{attribute 'qualified_only'}
// ------------------------------------------------------------------------- 
//  SRCI Robot Library                                                
// ------------------------------------------------------------------------- 
//                                                                           
//  Object:      RiState                                       
//  Author:      Thorsten Brach                                                
//  Date:        2024-06-01
//
//  Description:                                              
//   
//                                                                           
//  Copyright: 
//    (C) 2024 Thorsten Brach. All rights reserved                                                                                                                                            
//             Licensed under the MIT License.
//                                                                           
//  Disclaimer:                                                                           
//    This project is provided without any guarantee and can be used for   
//    private and commercial purposes. Any use is at the user’s 
//    own risk and responsibility.
//
// -------------------------------------------------------------------------
TYPE RiState :
(
  /// RI is not initialized
  NOT_INITIALIZED := 0,
  /// Initialization finished successfully
  INITIALIZED := 1,
  /// Data between RC and PLC has been synchronized
  SYNCHRONIZED := 2
)USINT;
END_TYPE

{attribute 'qualified_only'}
TYPE TelegramState :
(
  /// Default
  UNDEFINED := 0,
  /// Telegram control does not match the telegram state
  ERROR_161_TELEGRAM_CONTROL_MISMATCH_TELEGRAM_STATE := 161,
  /// Initialization lost for unknown reason. See message log after reinitializing
  ERROR_162_INIT_LOST_UNKNOWN := 162,
  /// Telegram length does not match the length provided in the communication interface.
  ERROR_163_TELEGRAM_LENGTH_MISMATCH := 163,
  /// Incompatible major SRCI version
  ERROR_164_SRCI_MAJOR_VERSION_INCOMPATIBLE := 164,
  /// Lifesign timeout
  ERROR_165_LIFESIGN_TIMEOUT := 165,
  /// The selected optional cyclic data does not fit in the given telegram size
  ERROR_166_CYCLIC_DATA_TOO_LARGE := 166,
  /// The robot interface was reset after being initialized
  ERROR_167_INTERFACE_WAS_RESET_AFTER_INIT := 167,
  /// Telegram sequence timeout
  ERROR_168_TELEGRAM_SEQ_TIMEOUT := 168,
  /// The telegram number changed after initialization
  ERROR_169_TELEGRAM_NO_CHANGED_AFTER_INIT := 169,
  /// Invalid AxesGroupID
  ERROR_170_AXESGROUP_ID_INVALID := 170,
  /// Telegram number is invalid. E.g. TwoSequences is only activated in one direction
  ERROR_171_TELEGRAM_NUMBER_INVALID := 171,
  /// Telegram Number is not supported
  ERROR_172_TELEGRAM_NUMBER_NOT_SUPPORTED := 172,
  /// Server connection lost
  ERROR_173_SERVER_CONNECTION_LOST := 173,
  /// The RC is currently not initialized but has state in the ACR
  READY_TO_RESUME := 253,
  /// The RC is currently not initialized and has no state in the ACR
  READY_FOR_INITIALIZATION := 254,
  /// The RC state is Initialized
  INITIALIZED := 255  
)USINT;
END_TYPE

{attribute 'qualified_only'}
// ------------------------------------------------------------------------- 
//  SRCI Robot Library                                                
// ------------------------------------------------------------------------- 
//                                                                           
//  Object:      AreaType                                       
//  Author:      Thorsten Brach                                                
//  Date:        2024-06-01
//
//  Description:                                              
//   
//                                                                           
//  Copyright: 
//    (C) 2024 Thorsten Brach. All rights reserved                                                                                                                                            
//             Licensed under the MIT License.
//                                                                           
//  Disclaimer:                                                                           
//    This project is provided without any guarantee and can be used for   
//    private and commercial purposes. Any use is at the user’s 
//    own risk and responsibility.
//
// -------------------------------------------------------------------------
TYPE AreaType :
(
  /// 0: Axes
  AXES := 0,
  /// 1: Box (default)
  BOX := 1,
  /// 2: Cylinder
  CYLINDER := 2,
  /// 3: Sphere (only DefinitionMode 1)
  SPHERE := 3
)USINT;
END_TYPE

{attribute 'qualified_only'}
// ------------------------------------------------------------------------- 
//  SRCI Robot Library                                                
// ------------------------------------------------------------------------- 
//                                                                           
//  Object:      AxesGroupParameterCmdEntries                                       
//  Author:      Thorsten Brach                                                
//  Date:        2024-06-01
//
//  Description:                                              
//   
//                                                                           
//  Copyright: 
//    (C) 2024 Thorsten Brach. All rights reserved                                                                                                                                            
//             Licensed under the MIT License.
//                                                                           
//  Disclaimer:                                                                           
//    This project is provided without any guarantee and can be used for   
//    private and commercial purposes. Any use is at the user’s 
//    own risk and responsibility.
//
// -------------------------------------------------------------------------
TYPE AxesGroupParameterCmdEntries :
(
  /// Handles multiple mechanisms required for operation of the interface
  RobotTask := 0, // No function code  
  /// Read robot-specific data from the RC
  ReadRobotData := 9002,  
  /// Enable/Disable robot into RA power state "Enabled"
  EnableRobot := 1,  
  /// Acknowledgement all pending errors
  GroupReset := 2,  
  /// Read the actual position – TCP: X…RZ + config/Turn, Joint: (J1…E6)
  ReadActualPosition := 3,
  /// Read the actual position cyclically
  ReadActualPositionCyclic := 4,   
  /// Read D-H-parameters of robot
  ReadDHParameter := 5,  
  /// Restart/reboot of the RC
  RestartController := 6,  
  /// Read actual TCP velocity
  ReadActualTCPVelocity := 7,  
  /// Login on RC from PLC
  UserLogin := 8,  
  /// Switch language of robot teach pendant from PLC
  SwitchLanguage := 9,  
  /// Reads and writes specific configuration parameters on RC that are required for the RI to work
  ExchangeConfiguration := 10,  
  /// Set active sequence
  SetSequence := 11,  
  /// Change actual speed override
  ChangeSpeedOverride := 12,  
  /// Read error codes of pending errors and move them into user data block "RobotData"
  ReadMessages := 13,  
  /// Read reference values of robot dynamics for path movement
  ReadRobotReferenceDynamics := 14,  
  /// Change configuration of selected user frame number
  WriteFrameData := 15,  
  /// Change configuration of selected tool number
  WriteToolData := 16,  
  /// Change configuration of selected payload number
  WriteLoadData := 17,  
  /// Write reference values of robot dynamics for path movement
  WriteRobotReferenceDynamics := 18,  
  /// Write default values of dynamic parameters used by move commands
  WriteRobotDefaultDynamics := 19,  
  /// Read default values of dynamic parameters used by move commands
  ReadRobotDefaultDynamics := 20,  
  /// Read content of selected user frame number
  ReadFrameData := 21,  
  /// Read content of selected tool number
  ReadToolData := 22,  
  /// Read content of selected payload number
  ReadLoadData := 23,  
  /// Read actual software limits of the axes Positive and negative Limit of Joint J1…J6, E1…E6
  ReadRobotSWLimits := 24,  
  /// Change robot limits of robot axes (degree)
  WriteRobotSWLimits := 25,  
  /// Switch operation mode of RC (Automatic External, T1 External, T2 External)
  SetOperationMode := 26,  
  /// Read configuration of defined work areas
  ReadWorkArea := 27,  
  /// Define work area
  WriteWorkArea := 28,  
  /// Enable/Disable work areas of RC and check if TCP is inside/outside of active work area
  ActivateWorkArea := 29,  
  /// Monitor enabled work areas
  MonitorWorkArea := 30,  
  /// Jog robot manually
  GroupJog := 31,  
  /// Move the TCP to an absolute cartesian position (linear interpolation)
  MoveLinearAbsolute := 32,  
  /// Move Joints to an absolute cartesian position (Absolute cartesian PTP) (Joint interpolated movement)
  MoveDirectAbsolute := 33,  
  /// Move all joints to an absolute joint position (Absolute Joint PTP)
  MoveAxesAbsolute := 34,  
  /// Abort actual movement and delete buffer
  GroupStop := 35,  
  /// Interrupt active movement, possible to continue movement
  GroupInterrupt := 36,  
  /// Continue interrupted path
  GroupContinue := 37,  
  /// Move the TCP relative to the actual cartesian position (linear interpolation)
  MoveLinearRelative := 38,  
  /// Move Joints relative to relative cartesian position (Relative cartesian PTP) (Joint interpolated movement)
  MoveDirectRelative := 39,  
  /// Move all joints relative to actual joint position (Relative Joint PTP)
  MoveAxesRelative := 40,  
  /// Return to path left during active interrupt
  ReturnToPrimary := 41,  
  /// Move the TCP to an absolute joint position (linear interpolation)
  MoveCircularAbsolute := 42,  
  /// Move the TCP relative to the actual cartesian position (circular interpolation)
  MoveCircularRelative := 43,  
  /// Move the TCP relative to a reference cartesian position (linear interpolation)
  MoveLinearOffset := 44,  
  /// Move the TCP relative to a reference cartesian position (PTPT interpolation)
  MoveDirectOffset := 45,  
  /// Set wait command between motion commands
  WaitTime := 46,  
  /// Linear Move to target position through auxiliary position defined by offset in all dimensions (movement to target position linear)
  MoveApproachLinear := 47,  
  /// Linear Move from actual position to destination through auxiliary position defined by offset in all dimensions (movement to target position linear)
  MoveDepartLinear := 48,  
  /// Direct Move to target position through auxiliary position defined by offset in all dimensions (movement to target posi tion PTP)
  MoveApproachDirect := 49,  
  /// Direct Move from actual position to destination through auxiliary position defined by offset in all dimensions (movement to the target position PTP)
  MoveDepartDirect := 50,  
  /// Move robot into contact with obstruction (mechanical Limit) and hold it in this position
  SearchHardstop := 51,  
  /// Move robot into contact with obstruction (mechanical Limit) and hold it in this position
  SearchHardstopJ := 52,  
  /// Command several interpolated movement of robot arm on linear paths from actual position
  MovePickPlaceLinear := 53,  
  /// Commands interpolated movement of robot arm on a partly undefined path from actual position
  MovePickPlaceDirect := 54,  
  /// Activate conveyor tracking mode
  ActivateConveyorTracking := 55,  
  /// Redefine tracking position for conveyor tracking
  RedefineTrackingPos := 56,  
  /// Synchronize robot with conveyor
  SyncToConveyor := 57,  
  /// Configure conveyor parameters
  ConfigureConveyor := 58,  
  /// Activate superimposed motion of TCP to defined motion
  MoveSuperImposed := 59,  
  /// Activate superimposed motion of TCP to defined motion
  MoveSuperImposedDynamic := 60,  
  /// Read digital input and output group of RC
  ReadDigitalInputs := 61,  
  /// Read digital output group of RC
  ReadDigitalOutputs := 62,  
  /// Write digital output group of RC
  WriteDigitalOutputs := 63,  
  /// Read integer values on RC
  ReadIntegers := 64,  
  /// Read real values on RC
  ReadReals := 65,  
  /// Write integer values on RC
  WriteIntegers := 66,  
  /// Write real values on RC
  WriteReals := 67,  
  /// Set trigger in defined position of path (L = Linear Path) (cartesian) switch periphery.
  MoveLinearCam := 68,  
  /// Set a trigger in a defined position of a path. (PTP)
  MoveDirectCam := 69,  
  /// Set a trigger in a defined position of a circular path
  MoveCircularCam := 70,  
  /// Read analog input of RC
  ReadAnalogInput := 71,  
  /// Read analog output of RC
  ReadAnalogOutput := 72,  
  /// Write analog output of RC
  WriteAnalogOutput := 73,  
  /// Capture trigger Position, measuring input
  MeasuringInput := 74,  
  /// Abort triggering of Position, measuring input
  AbortMeasuringInput := 75,  
  /// Trigger "Actions" based on I/O related events (e.g. change of DI’s state)
  SetTriggerRegister := 76,  
  /// Trigger "Actions" based on physical events (e.g. force limit reached)
  SetTriggerLimit := 77,  
  /// Trigger "Actions" based on physical events (e.g. force limit reached)
  SetTriggerUser := 78,  
  /// Trigger "Actions" based on incoming error event
  SetTriggerError := 79,  
  /// "Action" that initiates specified events when triggered
  ReactAtTrigger := 80,  
  /// Wait to process next command in sequence until trigger signal is received
  WaitForTrigger := 81,  
  /// Read specific parameter of the robot
  ReadSystemVariable := 82,  
  /// Change value of specific vendor parameter
  WriteSystemVariable := 83,  
  /// Calculate Forward Kinematic
  CalculateForwardKinematic := 84,  
  /// Calculate Inverse Kinematic
  CalculateInverseKinematic := 85,  
  /// Calculate cartesian position from existing cartesian position
  CalculateCartesianPosition := 86,  
  /// Calculate tool (TCP) with four-point method
  CalculateTool := 87,  
  /// Calculate frame with three-point method
  CalculateFrame := 88,  
  /// Cancel currently active move command and continue with the next buffered command
  ActivateNextCommand := 89,  
  /// Transform a defined position in space
  ShiftPosition := 90,  
  /// Trigger an action based on a motion-related parameter (e.g. progress of trajectory)
  SetTriggerMotion := 91,  
  /// Release robot arm’s brakes
  OpenBrake := 92,  
  /// Call subprogram stored in RC from PLC
  CallSubprogram := 93,  
  /// Writes cyclic data of called subprogram
  WriteCallSubprogramCyclic := 94,
  /// Reads cyclic data of called subprogram
  ReadCallSubprogramCyclic := 95,
  /// Stops an active subprogram
  StopSubprogram := 96,  
  /// Switch path mode between high and low accuracy
  PathAccuracyMode := 97,  
  /// Activate/Deactivate functionality to avoid singularities
  AvoidSingularity := 98,  
  /// Enables the RC to apply user-defined force/torque through RA’s TCP movement
  ForceControl := 99,  
  /// Commands specified reaction from RA when defined force/torque detected
  ForceLimit := 100,  
  /// Read actual force/torque at TCP
  ReadActualForce := 101,  
  /// Activate robot cycle brake test and give feedback to PLC
  BrakeTest := 102,  
  /// Push robot: Robot calculates opposite vector and moves slowly in that direction
  SoftSwitchTCP := 103,  
  /// Create spline on RC from positions stored in PLC
  CreateSpline := 104,  
  /// Delete spline previously created on RC
  DeleteSpline := 105,  
  /// Move spline previously created on RC
  MoveSpline := 106,  
  /// Create and move spline on RC simultaneously
  DynamicSpline := 107,  
  /// Automatic detection of load data
  LoadMeasurementAutomatic := 108,  
  /// Sequential detection of load data
  LoadMeasurementSequential := 109,  
  /// Turn on/off the collision detection
  CollisionDetection := 110,  
  /// Move the robot axes by hand
  FreeDrive := 111,  
  /// Measure the length of objects in the cartesian space, execution time for specified section of a job or signal output time of a specified signal
  UnitMeasurement := 112,
  /// Maximum entry
  MAX_ENTRY := 113   
)UINT;
END_TYPE

{attribute 'qualified_only'}
// ------------------------------------------------------------------------- 
//  SRCI Robot Library                                                
// ------------------------------------------------------------------------- 
//                                                                           
//  Object:      CmdType                                       
//  Author:      Thorsten Brach                                                
//  Date:        2024-06-01
//
//  Description:                                              
//   
//                                                                           
//  Copyright: 
//    (C) 2024 Thorsten Brach. All rights reserved                                                                                                                                            
//             Licensed under the MIT License.
//                                                                           
//  Disclaimer:                                                                           
//    This project is provided without any guarantee and can be used for   
//    private and commercial purposes. Any use is at the user’s 
//    own risk and responsibility.
//
// -------------------------------------------------------------------------
TYPE CmdType :
(
  /// Handles multiple mechanisms required for operation of the interface
  RobotTask := 0, // No function code  
  /// Read robot-specific data from the RC
  ReadRobotData := 9002,  
  /// Enable/Disable robot into RA power state "Enabled"
  EnableRobot := 1000,  
  /// Acknowledgement all pending errors
  GroupReset := 1001,  
  /// Read the actual position – TCP: X…RZ + config/Turn, Joint: (J1…E6)
  ReadActualPosition := 5100,
  /// Read the actual position cyclically
  ReadActualPositionCyclic := 1, // No function code  
  /// Read D-H-parameters of robot
  ReadDHParameter := 5101,  
  /// Restart/reboot of the RC
  RestartController := 1101,  
  /// Read actual TCP velocity
  ReadActualTCPVelocity := 5111,  
  /// Login on RC from PLC
  UserLogin := 1006,  
  /// Switch language of robot teach pendant from PLC
  SwitchLanguage := 1005,  
  /// Reads and writes specific configuration parameters on RC that are required for the RI to work
  ExchangeConfiguration := 9000,  
  /// Set active sequence
  SetSequence := 1004,  
  /// Change actual speed override
  ChangeSpeedOverride := 2000,  
  /// Read error codes of pending errors and move them into user data block "RobotData"
  ReadMessages := 9001,  
  /// Read reference values of robot dynamics for path movement
  ReadRobotReferenceDynamics := 5105,  
  /// Change configuration of selected user frame number
  WriteFrameData := 5200,  
  /// Change configuration of selected tool number
  WriteToolData := 5205,  
  /// Change configuration of selected payload number
  WriteLoadData := 5201,  
  /// Write reference values of robot dynamics for path movement
  WriteRobotReferenceDynamics := 5203,  
  /// Write default values of dynamic parameters used by move commands
  WriteRobotDefaultDynamics := 5202,  
  /// Read default values of dynamic parameters used by move commands
  ReadRobotDefaultDynamics := 5104,  
  /// Read content of selected user frame number
  ReadFrameData := 5102,  
  /// Read content of selected tool number
  ReadToolData := 5107,  
  /// Read content of selected payload number
  ReadLoadData := 5103,  
  /// Read actual software limits of the axes Positive and negative Limit of Joint J1…J6, E1…E6
  ReadRobotSWLimits := 5106,  
  /// Change robot limits of robot axes (degree)
  WriteRobotSWLimits := 5204,  
  /// Switch operation mode of RC (Automatic External, T1 External, T2 External)
  SetOperationMode := 1003,  
  /// Read configuration of defined work areas
  ReadWorkArea := 7502,  
  /// Define work area
  WriteWorkArea := 7503,  
  /// Enable/Disable work areas of RC and check if TCP is inside/outside of active work area
  ActivateWorkArea := 7500,  
  /// Monitor enabled work areas
  MonitorWorkArea := 7501,  
  /// Jog robot manually
  GroupJog := 2100,  
  /// Move the TCP to an absolute cartesian position (linear interpolation)
  MoveLinearAbsolute := 2103,  
  /// Move Joints to an absolute cartesian position (Absolute cartesian PTP) (Joint interpolated movement)
  MoveDirectAbsolute := 2102,  
  /// Move all joints to an absolute joint position (Absolute Joint PTP)
  MoveAxesAbsolute := 2101,  
  /// Abort actual movement and delete buffer
  GroupStop := 2003,  
  /// Interrupt active movement, possible to continue movement
  GroupInterrupt := 2002,  
  /// Continue interrupted path
  GroupContinue := 2001,  
  /// Move the TCP relative to the actual cartesian position (linear interpolation)
  MoveLinearRelative := 2110,  
  /// Move Joints relative to relative cartesian position (Relative cartesian PTP) (Joint interpolated movement)
  MoveDirectRelative := 2108,  
  /// Move all joints relative to actual joint position (Relative Joint PTP)
  MoveAxesRelative := 2105,  
  /// Return to path left during active interrupt
  ReturnToPrimary := 2104,  
  /// Move the TCP to an absolute joint position (linear interpolation)
  MoveCircularAbsolute := 2109,  
  /// Move the TCP relative to the actual cartesian position (circular interpolation)
  MoveCircularRelative := 2106,  
  /// Move the TCP relative to a reference cartesian position (linear interpolation)
  MoveLinearOffset := 2112,  
  /// Move the TCP relative to a reference cartesian position (PTPT interpolation)
  MoveDirectOffset := 2111,  
  /// Set wait command between motion commands
  WaitTime := 7005,  
  /// Linear Move to target position through auxiliary position defined by offset in all dimensions (movement to target position linear)
  MoveApproachLinear := 2201,  
  /// Linear Move from actual position to destination through auxiliary position defined by offset in all dimensions (movement to target position linear)
  MoveDepartLinear := 2203,  
  /// Direct Move to target position through auxiliary position defined by offset in all dimensions (movement to target posi tion PTP)
  MoveApproachDirect := 2200,  
  /// Direct Move from actual position to destination through auxiliary position defined by offset in all dimensions (movement to the target position PTP)
  MoveDepartDirect := 2202,  
  /// Move robot into contact with obstruction (mechanical Limit) and hold it in this position
  SearchHardstop := 2500,  
  /// Move robot into contact with obstruction (mechanical Limit) and hold it in this position
  SearchHardstopJ := 2501,  
  /// Command several interpolated movement of robot arm on linear paths from actual position
  MovePickPlaceLinear := 2205,  
  /// Commands interpolated movement of robot arm on a partly undefined path from actual position
  MovePickPlaceDirect := 2204,  
  /// Activate conveyor tracking mode
  ActivateConveyorTracking := 2300,  
  /// Redefine tracking position for conveyor tracking
  RedefineTrackingPos := 2302,  
  /// Synchronize robot with conveyor
  SyncToConveyor := 2303,  
  /// Configure conveyor parameters
  ConfigureConveyor := 2301,  
  /// Activate superimposed motion of TCP to defined motion
  MoveSuperImposed := 2502,  
  /// Activate superimposed motion of TCP to defined motion
  MoveSuperImposedDynamic := 2503,  
  /// Read digital input and output group of RC
  ReadDigitalInputs := 6100,  
  /// Read digital output group of RC
  ReadDigitalOutputs := 6101,  
  /// Write digital output group of RC
  WriteDigitalOutputs := 6104,  
  /// Read integer values on RC
  ReadIntegers := 6102,  
  /// Read real values on RC
  ReadReals := 6103,  
  /// Write integer values on RC
  WriteIntegers := 6105,  
  /// Write real values on RC
  WriteReals := 6106,  
  /// Set trigger in defined position of path (L = Linear Path) (cartesian) switch periphery.
  MoveLinearCam := 2402,  
  /// Set a trigger in a defined position of a path. (PTP)
  MoveDirectCam := 2401,  
  /// Set a trigger in a defined position of a circular path
  MoveCircularCam := 2400,  
  /// Read analog input of RC
  ReadAnalogInput := 6107,  
  /// Read analog output of RC
  ReadAnalogOutput := 6108,  
  /// Write analog output of RC
  WriteAnalogOutput := 6109,  
  /// Capture trigger Position, measuring input
  MeasuringInput := 6001,  
  /// Abort triggering of Position, measuring input
  AbortMeasuringInput := 6000,  
  /// Trigger "Actions" based on I/O related events (e.g. change of DI’s state)
  SetTriggerRegister := 3004,  
  /// Trigger "Actions" based on physical events (e.g. force limit reached)
  SetTriggerLimit := 3002,  
  /// Trigger "Actions" based on physical events (e.g. force limit reached)
  SetTriggerUser := 3005,  
  /// Trigger "Actions" based on incoming error event
  SetTriggerError := 3001,  
  /// "Action" that initiates specified events when triggered
  ReactAtTrigger := 3000,  
  /// Wait to process next command in sequence until trigger signal is received
  WaitForTrigger := 3006,  
  /// Read specific parameter of the robot
  ReadSystemVariable := 5109,  
  /// Change value of specific vendor parameter
  WriteSystemVariable := 5206,  
  /// Calculate Forward Kinematic
  CalculateForwardKinematic := 7203,  
  /// Calculate Inverse Kinematic
  CalculateInverseKinematic := 7204,  
  /// Calculate cartesian position from existing cartesian position
  CalculateCartesianPosition := 7200,  
  /// Calculate tool (TCP) with four-point method
  CalculateTool := 7202,  
  /// Calculate frame with three-point method
  CalculateFrame := 7201,  
  /// Cancel currently active move command and continue with the next buffered command
  ActivateNextCommand := 7000,  
  /// Transform a defined position in space
  ShiftPosition := 7205,  
  /// Trigger an action based on a motion-related parameter (e.g. progress of trajectory)
  SetTriggerMotion := 3003,  
  /// Release robot arm’s brakes
  OpenBrake := 7100,  
  /// Call subprogram stored in RC from PLC
  CallSubprogram := 7001,  
  /// Writes cyclic data of called subprogram
  WriteCallSubprogramCyclic := 2, // No function code
  /// Reads cyclic data of called subprogram
  ReadCallSubprogramCyclic := 3, // No function code
  /// Stops an active subprogram
  StopSubprogram := 7008,  
  /// Switch path mode between high and low accuracy
  PathAccuracyMode := 7401,  
  /// Activate/Deactivate functionality to avoid singularities
  AvoidSingularity := 7400,  
  /// Enables the RC to apply user-defined force/torque through RA’s TCP movement
  ForceControl := 7301,  
  /// Commands specified reaction from RA when defined force/torque detected
  ForceLimit := 7302,  
  /// Read actual force/torque at TCP
  ReadActualForce := 5110,  
  /// Activate robot cycle brake test and give feedback to PLC
  BrakeTest := 7101,  
  /// Push robot: Robot calculates opposite vector and moves slowly in that direction
  SoftSwitchTCP := 7300,  
  /// Create spline on RC from positions stored in PLC
  CreateSpline := 2600,  
  /// Delete spline previously created on RC
  DeleteSpline := 2601,  
  /// Move spline previously created on RC
  MoveSpline := 2603,  
  /// Create and move spline on RC simultaneously
  DynamicSpline := 2602,  
  /// Automatic detection of load data
  LoadMeasurementAutomatic := 7006,  
  /// Sequential detection of load data
  LoadMeasurementSequential := 7007,  
  /// Turn on/off the collision detection
  CollisionDetection := 7003,  
  /// Move the robot axes by hand
  FreeDrive := 7002,  
  /// Measure the length of objects in the cartesian space, execution time for specified section of a job or signal output time of a specified signal
  UnitMeasurement := 7004   
)UINT;
END_TYPE

{attribute 'qualified_only'}
// ------------------------------------------------------------------------- 
//  SRCI Robot Library                                                
// ------------------------------------------------------------------------- 
//                                                                           
//  Object:      ConveyorType                                       
//  Author:      Thorsten Brach                                                
//  Date:        2024-06-01
//
//  Description:                                              
//   
//                                                                           
//  Copyright: 
//    (C) 2024 Thorsten Brach. All rights reserved                                                                                                                                            
//             Licensed under the MIT License.
//                                                                           
//  Disclaimer:                                                                           
//    This project is provided without any guarantee and can be used for   
//    private and commercial purposes. Any use is at the user’s 
//    own risk and responsibility.
//
// -------------------------------------------------------------------------
TYPE ConveyorType :
(
  /// Linear Conveyor Tracking (default)
  LINEAR_CONVEYOR_TRACKING := 0,
  /// Circular Conveyor Tracking
  CIRCULAR_CONVEYOR_TRACKING := 1
)USINT;
END_TYPE

{attribute 'qualified_only'}
// ------------------------------------------------------------------------- 
//  SRCI Robot Library                                                
// ------------------------------------------------------------------------- 
//                                                                           
//  Object:      DataType                                       
//  Author:      Thorsten Brach                                                
//  Date:        2025-03-05
//
//  Description:                                              
//   
//                                                                           
//  Copyright: 
//    (C) 2025 Thorsten Brach. All rights reserved                                                                                                                                            
//             Licensed under the MIT License.
//                                                                           
//  Disclaimer:                                                                           
//    This project is provided without any guarantee and can be used for   
//    private and commercial purposes. Any use is at the user’s 
//    own risk and responsibility.
//
// -------------------------------------------------------------------------
TYPE DataType :
(
  /// BOOL
  TYPE_BOOL       := 1,
  /// BYTE        
  TYPE_BYTE       := 2,
  /// WORD        
  TYPE_WORD       := 3,
  /// DWORD       
  TYPE_DWORD      := 4,
  /// SINT        
  TYPE_SINT       := 5,
  /// USINT       
  TYPE_USINT      := 6,
  /// INT         
  TYPE_INT        := 7,
  /// UINT        
  TYPE_UINT       := 8,
  /// DINT        
  TYPE_DINT       := 9,
  /// UDINT       
  TYPE_UDINT      := 10,
  /// REAL        
  TYPE_REAL       := 11,
  /// CHAR
  TYPE_CHAR       := 12,
  /// CHAR_ARRAY
  TYPE_CHAR_ARRAY := 13  
)USINT;
END_TYPE

{attribute 'qualified_only'}
// ------------------------------------------------------------------------- 
//  SRCI Robot Library                                                
// ------------------------------------------------------------------------- 
//                                                                           
//  Object:      MessageType                                       
//  Author:      Thorsten Brach                                                
//  Date:        2024-06-01
//
//  Description:                                              
//   
//                                                                           
//  Copyright: 
//    (C) 2024 Thorsten Brach. All rights reserved                                                                                                                                            
//             Licensed under the MIT License.
//                                                                           
//  Disclaimer:                                                                           
//    This project is provided without any guarantee and can be used for   
//    private and commercial purposes. Any use is at the user’s 
//    own risk and responsibility.
//
// -------------------------------------------------------------------------
TYPE MessageType :
(
  /// RI related messages
  RI := 1,
  /// RC related messages
  RC := 2,
  /// RA related messages
  RA := 3, 
  /// Command related messages
  CMD := 4 
)USINT;
END_TYPE

{attribute 'qualified_only'}
// ------------------------------------------------------------------------- 
//  SRCI Robot Library                                                
// ------------------------------------------------------------------------- 
//                                                                           
//  Object:      ReferenceType                                       
//  Author:      Thorsten Brach                                                
//  Date:        2024-06-01
//
//  Description:                                              
//   
//                                                                           
//  Copyright: 
//    (C) 2024 Thorsten Brach. All rights reserved                                                                                                                                            
//             Licensed under the MIT License.
//                                                                           
//  Disclaimer:                                                                           
//    This project is provided without any guarantee and can be used for   
//    private and commercial purposes. Any use is at the user’s 
//    own risk and responsibility.
//
// -------------------------------------------------------------------------
TYPE ReferenceType :
(
  /// Distance is applied in the Tool coordinate system. 
  /// The setting of the parameter FrameNo will be ignored.
  TOOL  := 0,
  /// Distance is applied in the Frame coordinate system.
  /// The settings of the ToolNo are also effective and must be considered. 
  FRAME := 1
)USINT;
END_TYPE

{attribute 'qualified_only'}
// ------------------------------------------------------------------------- 
//  SRCI Robot Library                                                
// ------------------------------------------------------------------------- 
//                                                                           
//  Object:      UnitType                                       
//  Author:      Thorsten Brach                                                
//  Date:        2024-06-01
//
//  Description:                                              
//   
//                                                                           
//  Copyright: 
//    (C) 2024 Thorsten Brach. All rights reserved                                                                                                                                            
//             Licensed under the MIT License.
//                                                                           
//  Disclaimer:                                                                           
//    This project is provided without any guarantee and can be used for   
//    private and commercial purposes. Any use is at the user’s 
//    own risk and responsibility.
//
// -------------------------------------------------------------------------
TYPE UnitType :
(
  /// Volt
  VOLT   := 0,
  /// Ampere
  AMPERE := 1
)USINT;
END_TYPE

{attribute 'pack_mode' := '1'} 
// ------------------------------------------------------------------------- 
//  SRCI Robot Library                                                
// ------------------------------------------------------------------------- 
//                                                                           
//  Object:      AbortMeasuringInputOutCmd                                       
//  Author:      Thorsten Brach                                                
//  Date:        2024-06-21
//
//  Description:                                              
//   
//                                                                           
//  Copyright: 
//    (C) 2024 Thorsten Brach. All rights reserved                                                                                                                                            
//             Licensed under the MIT License.
//                                                                           
//  Disclaimer:                                                                           
//    This project is provided without any guarantee and can be used for   
//    private and commercial purposes. Any use is at the user’s 
//    own risk and responsibility.
//
// -------------------------------------------------------------------------
TYPE AbortMeasuringInputOutCmd :
STRUCT
END_STRUCT
END_TYPE

{attribute 'pack_mode' := '1'} 
// ------------------------------------------------------------------------- 
//  SRCI Robot Library                                                
// ------------------------------------------------------------------------- 
//                                                                           
//  Object:      AbortMeasuringInputParCmd                                       
//  Author:      Thorsten Brach                                                
//  Date:        2024-06-21
//
//  Description:                                              
//   
//                                                                           
//  Copyright: 
//    (C) 2024 Thorsten Brach. All rights reserved                                                                                                                                            
//             Licensed under the MIT License.
//                                                                           
//  Disclaimer:                                                                           
//    This project is provided without any guarantee and can be used for   
//    private and commercial purposes. Any use is at the user’s 
//    own risk and responsibility.
//
// -------------------------------------------------------------------------
TYPE AbortMeasuringInputParCmd :
STRUCT
  /// Define an active measurement that is to be aborted.
  /// •  0: Abort all existing measurement
  /// • >0: Abort the measurement with the specific MeasuringID
  MeasuringID        : UINT;
END_STRUCT
END_TYPE

{attribute 'pack_mode' := '1'} 
// ------------------------------------------------------------------------- 
//  SRCI Robot Library                                                
// ------------------------------------------------------------------------- 
//                                                                           
//  Object:      AbortMeasuringInputRecvData                                       
//  Author:      Thorsten Brach                                                
//  Date:        2024-06-21
//
//  Description:                                              
//   
//                                                                           
//  Copyright: 
//    (C) 2024 Thorsten Brach. All rights reserved                                                                                                                                            
//             Licensed under the MIT License.
//                                                                           
//  Disclaimer:                                                                           
//    This project is provided without any guarantee and can be used for   
//    private and commercial purposes. Any use is at the user’s 
//    own risk and responsibility.
//
// -------------------------------------------------------------------------
TYPE AbortMeasuringInputRecvData EXTENDS RspHeader :
STRUCT
END_STRUCT
END_TYPE

{attribute 'pack_mode' := '1'}
// ------------------------------------------------------------------------- 
//  SRCI Robot Library                                                
// ------------------------------------------------------------------------- 
//                                                                           
//  Object:      AbortMeasuringInputSendData                                       
//  Author:      Thorsten Brach                                                
//  Date:        2024-06-21
//
//  Description:                                              
//   
//                                                                           
//  Copyright: 
//    (C) 2024 Thorsten Brach. All rights reserved                                                                                                                                            
//             Licensed under the MIT License.
//                                                                           
//  Disclaimer:                                                                           
//    This project is provided without any guarantee and can be used for   
//    private and commercial purposes. Any use is at the user’s 
//    own risk and responsibility.
//
// -------------------------------------------------------------------------
TYPE AbortMeasuringInputSendData EXTENDS CmdHeader:   
STRUCT
  /// Define an active measurement that is to be aborted.
  /// •  0: Abort all existing measurement
  /// • >0: Abort the measurement with the specific MeasuringID
  MeasuringID        : UINT;
END_STRUCT
END_TYPE

{attribute 'pack_mode' := '1'} 
// ------------------------------------------------------------------------- 
//  SRCI Robot Library                                                
// ------------------------------------------------------------------------- 
//                                                                           
//  Object:      ActivateNextCommandOutCmd                                       
//  Author:      Thorsten Brach                                                
//  Date:        2024-06-01
//
//  Description:                                              
//   
//                                                                           
//  Copyright: 
//             Licensed under the MIT License.
//    (C) 2024 Thorsten Brach. All rights reserved                                                                                                                                            
//                                                                           
//  Disclaimer:                                                                           
//    This project is provided without any guarantee and can be used for   
//    private and commercial purposes. Any use is at the user’s 
//    own risk and responsibility.
//
// -------------------------------------------------------------------------
TYPE ActivateNextCommandOutCmd :
STRUCT
  /// Unique system-generated ID of the "Action" when the function is triggered.
  /// • >0: The "Action" is started by the trigger function with identical FollowID.
  /// • <0: The "Action" is stopped by the trigger function with identical FollowID.
  /// For more information see chapter 5.5.12.4 EmitterID, ListenerID, FollowID and OriginID
  OriginID           : INT;
  /// Relates to ListenerID >0
  /// Number of successful trigger -based command invocations
  /// For more information refer to chapter 5.5.12.4.
  InvocationCounter  : USINT;
END_STRUCT
END_TYPE

{attribute 'pack_mode' := '1'} 
// ------------------------------------------------------------------------- 
//  SRCI Robot Library                                                
// ------------------------------------------------------------------------- 
//                                                                           
//  Object:      ActivateNextCommandParCmd                                       
//  Author:      Thorsten Brach                                                
//  Date:        2024-06-01
//
//  Description:                                              
//   
//                                                                           
//  Copyright: 
//    (C) 2024 Thorsten Brach. All rights reserved                                                                                                                                            
//             Licensed under the MIT License.
//                                                                           
//  Disclaimer:                                                                           
//    This project is provided without any guarantee and can be used for   
//    private and commercial purposes. Any use is at the user’s 
//    own risk and responsibility.
//
// -------------------------------------------------------------------------
TYPE ActivateNextCommandParCmd :
STRUCT
  /// ID of the trigger function that may be triggered:
  /// • 0: Immediately (default). - Start executing THIS function immediately.
  /// • >0: Triggero Start executing when the trigger function with the identical EmitterID is called.
  /// For more information see chapter 5.5.12.4.
  ListenerID     : SINT;
END_STRUCT
END_TYPE

{attribute 'pack_mode' := '1'} 
// ------------------------------------------------------------------------- 
//  SRCI Robot Library                                                
// ------------------------------------------------------------------------- 
//                                                                           
//  Object:      ActivateNextCommandRecvData                                       
//  Author:      Thorsten Brach                                                
//  Date:        2024-06-01
//
//  Description:                                              
//   
//                                                                           
//  Copyright: 
//    (C) 2024 Thorsten Brach. All rights reserved                                                                                                                                            
//             Licensed under the MIT License.
//                                                                           
//  Disclaimer:                                                                           
//    This project is provided without any guarantee and can be used for   
//    private and commercial purposes. Any use is at the user’s 
//    own risk and responsibility.
//
// -------------------------------------------------------------------------
TYPE ActivateNextCommandRecvData EXTENDS RspHeader :
STRUCT
  /// Relates to ListenerID >0
  /// Number of successful trigger -based command invocations
  /// For more information refer to chapter 5.5.12.4.
  InvocationCounter  : USINT;
  /// Reserve
  Reserve            : SINT;
  /// Unique system-generated ID of the "Action" when the function is triggered.
  /// • >0: The "Action" is started by the trigger function with identical FollowID.
  /// • <0: The "Action" is stopped by the trigger function with identical FollowID.
  /// For more information see chapter 5.5.12.4 EmitterID, ListenerID, FollowID and OriginID
  OriginID           : INT;
END_STRUCT
END_TYPE

{attribute 'pack_mode' := '1'}
// ------------------------------------------------------------------------- 
//  SRCI Robot Library                                                
// ------------------------------------------------------------------------- 
//                                                                           
//  Object:      ActivateNextCommandParCmd                                       
//  Author:      Thorsten Brach                                                
//  Date:        2024-06-01
//
//  Description:                                              
//   
//                                                                           
//  Copyright: 
//    (C) 2024 Thorsten Brach. All rights reserved                                                                                                                                            
//             Licensed under the MIT License.
//                                                                           
//  Disclaimer:                                                                           
//    This project is provided without any guarantee and can be used for   
//    private and commercial purposes. Any use is at the user’s 
//    own risk and responsibility.
//
// -------------------------------------------------------------------------
TYPE ActivateNextCommandSendData EXTENDS CmdHeader:   
STRUCT  
  /// ID of Action that will be executed when this command is active
  /// • >0: Start Action        - Start executing the Action function with the identical ListenerID.
  /// • <0: Stop Action         - Stop executing the Action function with the identical ListenerID.
  /// •  0: Undefined (default) - If no EmitterID is defined, the function returns an error message
  /// For more information see chapter 5.5.12.4
  EmitterID  : ARRAY[0..3] OF SINT;  
  /// ID of the trigger function that may be triggered:
  /// • 0: Immediately (default). - Start executing THIS function immediately.
  /// • >0: Triggero Start executing when the trigger function with the identical EmitterID is called.
  /// For more information see chapter 5.5.12.4.
  ListenerID : SINT;
  /// Reserve
  Reserve    : BYTE;
END_STRUCT
END_TYPE

{attribute 'pack_mode' := '1'} 
// ------------------------------------------------------------------------- 
//  SRCI Robot Library                                                
// ------------------------------------------------------------------------- 
//                                                                           
//  Object:      AvoidSingularityOutCmd                                       
//  Author:      Thorsten Brach                                                
//  Date:        2024-06-22
//
//  Description:                                              
//   
//                                                                           
//  Copyright: 
//    (C) 2024 Thorsten Brach. All rights reserved                                                                                                                                            
//             Licensed under the MIT License.
//                                                                           
//  Disclaimer:                                                                           
//    This project is provided without any guarantee and can be used for   
//    private and commercial purposes. Any use is at the user’s 
//    own risk and responsibility.
//
// -------------------------------------------------------------------------
TYPE AvoidSingularityOutCmd :
STRUCT
END_STRUCT
END_TYPE

{attribute 'pack_mode' := '1'} 
// ------------------------------------------------------------------------- 
//  SRCI Robot Library                                                
// ------------------------------------------------------------------------- 
//                                                                           
//  Object:      AvoidSingularityParCmd                                       
//  Author:      Thorsten Brach                                                
//  Date:        2024-06-22
//
//  Description:                                              
//   
//                                                                           
//  Copyright: 
//    (C) 2024 Thorsten Brach. All rights reserved                                                                                                                                            
//             Licensed under the MIT License.
//                                                                           
//  Disclaimer:                                                                           
//    This project is provided without any guarantee and can be used for   
//    private and commercial purposes. Any use is at the user’s 
//    own risk and responsibility.
//
// -------------------------------------------------------------------------
TYPE AvoidSingularityParCmd :
STRUCT
  /// Define in which way the singularity should be avoided
  Mode : SingularityAvoidanceMode; 
END_STRUCT
END_TYPE

{attribute 'pack_mode' := '1'} 
// ------------------------------------------------------------------------- 
//  SRCI Robot Library                                                
// ------------------------------------------------------------------------- 
//                                                                           
//  Object:      AvoidSingularityRecvData                                       
//  Author:      Thorsten Brach                                                
//  Date:        2024-06-22
//
//  Description:                                              
//   
//                                                                           
//  Copyright: 
//    (C) 2024 Thorsten Brach. All rights reserved                                                                                                                                            
//             Licensed under the MIT License.
//                                                                           
//  Disclaimer:                                                                           
//    This project is provided without any guarantee and can be used for   
//    private and commercial purposes. Any use is at the user’s 
//    own risk and responsibility.
//
// -------------------------------------------------------------------------
TYPE AvoidSingularityRecvData EXTENDS RspHeader :
STRUCT
  /// TRUE when robot is set to RA power state "Enabled".
  Enabled : BOOL;
END_STRUCT
END_TYPE

{attribute 'pack_mode' := '1'}
// ------------------------------------------------------------------------- 
//  SRCI Robot Library                                                
// ------------------------------------------------------------------------- 
//                                                                           
//  Object:      AvoidSingularitySendData                                       
//  Author:      Thorsten Brach                                                
//  Date:        2024-06-22
//
//  Description:                                              
//   
//                                                                           
//  Copyright: 
//    (C) 2024 Thorsten Brach. All rights reserved                                                                                                                                            
//             Licensed under the MIT License.
//                                                                           
//  Disclaimer:                                                                           
//    This project is provided without any guarantee and can be used for   
//    private and commercial purposes. Any use is at the user’s 
//    own risk and responsibility.
//
// -------------------------------------------------------------------------
TYPE AvoidSingularitySendData EXTENDS CmdHeader: 
STRUCT
  /// Set TRUE to activate avoid singularity mode
  Enable : BOOL;
  /// Define in which way the singularity should be avoided
  Mode   : SingularityAvoidanceMode;
END_STRUCT
END_TYPE

{attribute 'pack_mode' := '1'} 
// ------------------------------------------------------------------------- 
//  SRCI Robot Library                                                
// ------------------------------------------------------------------------- 
//                                                                           
//  Object:      BrakeTestOutCmd                                       
//  Author:      Thorsten Brach                                                
//  Date:        2024-06-01
//
//  Description:                                              
//   
//                                                                           
//  Copyright: 
//    (C) 2024 Thorsten Brach. All rights reserved                                                                                                                                            
//             Licensed under the MIT License.
//                                                                           
//  Disclaimer:                                                                           
//    This project is provided without any guarantee and can be used for   
//    private and commercial purposes. Any use is at the user’s 
//    own risk and responsibility.
//
// -------------------------------------------------------------------------
TYPE BrakeTestOutCmd :
STRUCT
  /// Indicates the result of the brake test of the robot axes related to the brake test.
  /// • TRUE: The brake test has been realized successfully.
  /// • FALSE: The brake test failed. 
  /// See Table 6-735 for bit assignment.
  RobotAxesStatus    : RobotAxesFlags;
  /// Indicates the result of the brake test of the external robot axes related to the brake test.
  /// • TRUE: The brake test has been realized successfully.
  /// • FALSE: The brake test failed.
  /// See Table 6-735 for bit assignment.
  ExternalAxesStatus : ExternalAxesFlags;
  /// Indicates the warning messages availability related to the brake functionality of the robot axes reported by the RC.
  /// • TRUE: One or more warning messages are available.
  /// • FALSE: No warning message is available.
  /// See Table 6-735 for bit assignment.
  RobotAxesWarning   : RobotAxesFlags;
  /// Indicates the warning messages availability related to the brake functionality of the external robot axis reported by the RC.
  /// • TRUE: One or more warning messages are available.
  /// • FALSE: No warning message is available.
  /// See Table 6-735 for bit assignment.
  ExternalAxesWarning: ExternalAxesFlags;
END_STRUCT
END_TYPE

{attribute 'pack_mode' := '1'} 
// ------------------------------------------------------------------------- 
//  SRCI Robot Library                                                
// ------------------------------------------------------------------------- 
//                                                                           
//  Object:      BrakeTestParCmd                                       
//  Author:      Thorsten Brach                                                
//  Date:        2024-06-01
//
//  Description:                                              
//   
//                                                                           
//  Copyright: 
//    (C) 2024 Thorsten Brach. All rights reserved                                                                                                                                            
//             Licensed under the MIT License.
//                                                                           
//  Disclaimer:                                                                           
//    This project is provided without any guarantee and can be used for   
//    private and commercial purposes. Any use is at the user’s 
//    own risk and responsibility.
//
// -------------------------------------------------------------------------
TYPE BrakeTestParCmd :
STRUCT
  /// Defines which of the robot axis should be activated for the brake test.
  /// • TRUE (default): Axis activated.
  /// • FALSE: Axis deactivated.
  /// See Table 6-735 for bit assignment.
  RobotAxesActive    : RobotAxesFlags;
  /// Defines which of the external robot axis should be activated for the brake test.
  /// • TRUE: Axis activated.
  /// • FALSE (default): Axis deactivated.
  /// See Table 6-735 for bit assignment.   
  ExternalAxesActive : ExternalAxesFlags;
END_STRUCT
END_TYPE

{attribute 'pack_mode' := '1'} 
// ------------------------------------------------------------------------- 
//  SRCI Robot Library                                                
// ------------------------------------------------------------------------- 
//                                                                           
//  Object:      BrakeTestRecvData                                       
//  Author:      Thorsten Brach                                                
//  Date:        2024-06-01
//
//  Description:                                              
//   
//                                                                           
//  Copyright: 
//    (C) 2024 Thorsten Brach. All rights reserved                                                                                                                                            
//             Licensed under the MIT License.
//                                                                           
//  Disclaimer:                                                                           
//    This project is provided without any guarantee and can be used for   
//    private and commercial purposes. Any use is at the user’s 
//    own risk and responsibility.
//
// -------------------------------------------------------------------------
TYPE BrakeTestRecvData EXTENDS RspHeader :
STRUCT
  /// Indicates the result of the brake test of the robot axes related to the brake test.
  /// • TRUE: The brake test has been realized successfully.
  /// • FALSE: The brake test failed. 
  /// See Table 6-735 for bit assignment.
  RobotAxesStatus    : BYTE;
  /// Indicates the result of the brake test of the external robot axes related to the brake test.
  /// • TRUE: The brake test has been realized successfully.
  /// • FALSE: The brake test failed.
  /// See Table 6-735 for bit assignment.
  ExternalAxesStatus : BYTE;
  /// Indicates the warning messages availability related to the brake functionality of the robot axes reported by the RC.
  /// • TRUE: One or more warning messages are available.
  /// • FALSE: No warning message is available.
  /// See Table 6-735 for bit assignment.
  RobotAxesWarning   : BYTE;
  /// Indicates the warning messages availability related to the brake functionality of the external robot axis reported by the RC.
  /// • TRUE: One or more warning messages are available.
  /// • FALSE: No warning message is available.
  /// See Table 6-735 for bit assignment.
  ExternalAxesWarning: BYTE;
END_STRUCT
END_TYPE

{attribute 'pack_mode' := '1'}
// ------------------------------------------------------------------------- 
//  SRCI Robot Library                                                
// ------------------------------------------------------------------------- 
//                                                                           
//  Object:      BrakeTestSendData                                       
//  Author:      Thorsten Brach                                                
//  Date:        2024-06-01
//
//  Description:                                              
//   
//                                                                           
//  Copyright: 
//    (C) 2024 Thorsten Brach. All rights reserved                                                                                                                                            
//             Licensed under the MIT License.
//                                                                           
//  Disclaimer:                                                                           
//    This project is provided without any guarantee and can be used for   
//    private and commercial purposes. Any use is at the user’s 
//    own risk and responsibility.
//
// -------------------------------------------------------------------------
TYPE BrakeTestSendData EXTENDS CmdHeader:   
STRUCT
  /// Defines which of the robot axis should be activated for the brake test.
  /// • TRUE (default): Axis activated.
  /// • FALSE: Axis deactivated.
  /// See Table 6-735 for bit assignment.
  RobotAxesActive    : BYTE;
  /// Defines which of the external robot axis should be activated for the brake test.
  /// • TRUE: Axis activated.
  /// • FALSE (default): Axis deactivated.
  /// See Table 6-735 for bit assignment.   
  ExternalAxesActive : BYTE; 
END_STRUCT
END_TYPE

{attribute 'pack_mode' := '1'} 
// ------------------------------------------------------------------------- 
//  SRCI Robot Library                                                
// ------------------------------------------------------------------------- 
//                                                                           
//  Object:      CallSubprogramOutCmd                                       
//  Author:      Thorsten Brach                                                
//  Date:        2024-08-03
//
//  Description:                                              
//   
//                                                                           
//  Copyright: 
//    (C) 2024 Thorsten Brach. All rights reserved                                                                                                                                            
//             Licensed under the MIT License.
//                                                                           
//  Disclaimer:                                                                           
//    This project is provided without any guarantee and can be used for   
//    private and commercial purposes. Any use is at the user’s 
//    own risk and responsibility.
//
// -------------------------------------------------------------------------
TYPE CallSubprogramOutCmd :
STRUCT
  /// Unique, system-generated ID of the instance of CallSubprogram. 
  /// Can be used to specifically stop instance of a subprogram via the function Stop Subprogram (chapter 6.5.21) 
  /// if multiinstancing  is supported by RC 
  InstanceID         : DINT; 
  /// Unique system-generated ID of the "Action" when the function is triggered.
  /// • >0: The "Action" is started by the trigger function with identical FollowID.
  /// • <0: The "Action" is stopped by the trigger function with identical FollowID.
  /// For more information see chapter 5.5.12.4 EmitterID, ListenerID, FollowID and OriginID
  OriginID           : INT;
  /// Relates to ListenerID >0
  /// Number of successful trigger -based command invocations
  /// For more information refer to chapter 5.5.12.4.
  InvocationCounter  : USINT;
  /// The requested subprogram on the RC is in progress. Movement of the axes trough this subprogram is possible.
  InProgress         : BOOL;
  /// Acyclic output parameters of the subprogram Array length adjusts to transmitted data (max 190 bytes)
  ReturnData         : ARRAY[0..RobotLibraryParameter.SUB_PROGRAM_DATA_MAX] OF BYTE;
END_STRUCT
END_TYPE

{attribute 'pack_mode' := '1'} 
// ------------------------------------------------------------------------- 
//  SRCI Robot Library                                                
// ------------------------------------------------------------------------- 
//                                                                           
//  Object:      CallSubprogramParCmd                                       
//  Author:      Thorsten Brach                                                
//  Date:        2024-08-03
//
//  Description:                                              
//   
//                                                                           
//  Copyright: 
//    (C) 2024 Thorsten Brach. All rights reserved                                                                                                                                            
//             Licensed under the MIT License.
//                                                                           
//  Disclaimer:                                                                           
//    This project is provided without any guarantee and can be used for   
//    private and commercial purposes. Any use is at the user’s 
//    own risk and responsibility.
//
// -------------------------------------------------------------------------
TYPE CallSubprogramParCmd :
STRUCT
  /// Program number of the subprogram in the RC
  JobID          : UINT;
  /// ID of associated trigger function:
  /// • 0: No Trigger (default) - No trigger related behavior
  /// • >0: Triggero - Start executing when the trigger function with the identical EmitterID is triggered.
  /// Always positive.
  /// For more information, see chapter 5.5.12 Triggers
  ListenerID     : SINT;
  /// Acyclic input parameters of the subprogram Array length adjusts to transmitted data (max 190 bytes)
  Data           : ARRAY[0..RobotLibraryParameter.SUB_PROGRAM_DATA_MAX] OF BYTE;
END_STRUCT
END_TYPE

{attribute 'pack_mode' := '1'} 
// ------------------------------------------------------------------------- 
//  SRCI Robot Library                                                
// ------------------------------------------------------------------------- 
//                                                                           
//  Object:      CallSubprogramRecvData                                       
//  Author:      Thorsten Brach                                                
//  Date:        2024-08-03
//
//  Description:                                              
//   
//                                                                           
//  Copyright: 
//    (C) 2024 Thorsten Brach. All rights reserved                                                                                                                                            
//             Licensed under the MIT License.
//                                                                           
//  Disclaimer:                                                                           
//    This project is provided without any guarantee and can be used for   
//    private and commercial purposes. Any use is at the user’s 
//    own risk and responsibility.
//
// -------------------------------------------------------------------------
TYPE CallSubprogramRecvData EXTENDS RspHeader :
STRUCT
  /// Relates to ListenerID >0
  /// Number of successful trigger-based command invocations - For more information refer TO chapter 5.5.12.4
  InvocationCounter : USINT;  
  /// Reserve
  Reserve           : SINT;
  /// Unique system-generated ID of the "Action" when the function is triggered.
  /// • >0: The "Action" is started by the trigger funcrion with identical FollowID.
  /// • <0: The "Action" is stopped by the trigger function with identical FollowID.
  /// For more information see chapter 5.5.12.4 EmitterID, ListenerID, FollowID and OriginID
  OriginID          : INT;
  /// Percentage of already traversed distance of current job.
  /// If not supported : • -1
  Progress          : UINT;
  /// The requested subprogram on the RC is in progress. Movement of the axes trough this subprogram is possible.
  InProgress        : BOOL;
  /// Acyclic output parameters of the subprogram Array length adjusts to transmitted data (max 190 bytes)
  ReturnData        : ARRAY[0..RobotLibraryParameter.SUB_PROGRAM_DATA_MAX] OF BYTE;  
END_STRUCT
END_TYPE

{attribute 'pack_mode' := '1'}
// ------------------------------------------------------------------------- 
//  SRCI Robot Library                                                
// ------------------------------------------------------------------------- 
//                                                                           
//  Object:      CallSubprogramSendData                                       
//  Author:      Thorsten Brach                                                
//  Date:        2024-08-03
//
//  Description:                                              
//   
//                                                                           
//  Copyright: 
//    (C) 2024 Thorsten Brach. All rights reserved                                                                                                                                            
//             Licensed under the MIT License.
//                                                                           
//  Disclaimer:                                                                           
//    This project is provided without any guarantee and can be used for   
//    private and commercial purposes. Any use is at the user’s 
//    own risk and responsibility.
//
// -------------------------------------------------------------------------
TYPE CallSubprogramSendData EXTENDS CmdHeader: 
STRUCT
  /// ID of Action that will be executed when this command is active
  /// • >0: Start Action - Start executing the Action function with the identical ListenerID.
  /// • <0: Stop Action  -  Stop executing the Action function with the identical ListenerID.
  /// • 0: No trigger (default)-  If no EmitterID is defined, the function will not trigger any Action during its execution
  /// For more information see section Triggers of this chapter or chapter 5.5.12.4.
  EmitterID          : ARRAY [0..3] OF SINT;  
  /// ID of associated trigger function:
  /// • 0: No Trigger (default) - No trigger related behavior
  /// • >0: Triggero - Start executing when the trigger function with the identical EmitterID is triggered.
  /// Always positive.
  /// For more information, see chapter 5.5.12 Triggers
  ListenerID        : SINT;
  /// Reserve
  Reserve           : BYTE;
  /// Program number of the subprogram in the RC
  JobID             : UINT;
  /// Acyclic input parameters of the subprogram Array length adjusts to transmitted data (max 190 bytes)
  Data              : ARRAY[0..RobotLibraryParameter.SUB_PROGRAM_DATA_MAX] OF BYTE;
END_STRUCT
END_TYPE

{attribute 'pack_mode' := '1'} 
// ------------------------------------------------------------------------- 
//  SRCI Robot Library                                                
// ------------------------------------------------------------------------- 
//                                                                           
//  Object:      CollisionDetectionOutCmd                                       
//  Author:      Thorsten Brach                                                
//  Date:        2024-06-22
//
//  Description:                                              
//   
//                                                                           
//  Copyright: 
//    (C) 2024 Thorsten Brach. All rights reserved                                                                                                                                            
//             Licensed under the MIT License.
//                                                                           
//  Disclaimer:                                                                           
//    This project is provided without any guarantee and can be used for   
//    private and commercial purposes. Any use is at the user’s 
//    own risk and responsibility.
//
// -------------------------------------------------------------------------
TYPE CollisionDetectionOutCmd :
STRUCT
END_STRUCT
END_TYPE

{attribute 'pack_mode' := '1'} 
// ------------------------------------------------------------------------- 
//  SRCI Robot Library                                                
// ------------------------------------------------------------------------- 
//                                                                           
//  Object:      CollisionDetectionParCmd                                       
//  Author:      Thorsten Brach                                                
//  Date:        2024-06-22
//
//  Description:                                              
//   
//                                                                           
//  Copyright: 
//    (C) 2024 Thorsten Brach. All rights reserved                                                                                                                                            
//             Licensed under the MIT License.
//                                                                           
//  Disclaimer:                                                                           
//    This project is provided without any guarantee and can be used for   
//    private and commercial purposes. Any use is at the user’s 
//    own risk and responsibility.
//
// -------------------------------------------------------------------------
TYPE CollisionDetectionParCmd :
STRUCT
  /// Processing mode
  ProcessingMode     : ProcessingMode;
  ///  Defines the robot behavior after detecting the collision (at least one option must be supported):
  ReactionMode       : CollisionReactionMode;
  /// Set TRUE to activate and FALSE to deactivate "CollisionDetection".
  /// Default: TRUE
  ActivateMonitoring : BOOL;
  /// Defines the type of threshold setting (at least one option must be supported)
  ThresholdMode      : ThresholdMode;
  /// Defines the level of sensitivity of all axes.
  /// • 0..99: Sensitivity lower than robot vendor default. 
  ///          At minimum value "0" there is no sensitivity. The lower the value, the lower the sensitivity at the collision detection.
  /// • 100 (default): The value is aligned with the robot vendor-specific default value.
  /// • 101..200: Sensitivity higher than robot vendor default. At maximum value "200" highest possible sensitivity at the collision detection.
  Sensitivity        : REAL;
  /// Defines the level of sensitivity of the respective axis.
  /// Values:
  /// • 0..99: Sensitivity lower than robot vendor default. At minimum value "0" there is no sensitivity and collision detection for the respective axis. 
  ///          The lower the value, the lower the sensitivity at the collision detection.
  /// • 100 (default): The value is aligned with the robot vendor-specific default value.
  /// • 101..200: Sensitivity higher than robot vendor default. At maximum value "200" highest possible sensitivity at the collision detection.
  /// Index:
  /// • [0]: J1 First joint of the robot.
  /// • [1]: J2 Second joint of the robot.
  /// • [2] J3 Third joint of the robot.
  /// • [3] J4 Forth joint of the robot.
  /// • [4] J5 Fifth joint of the robot.
  /// • [5] J6 Six joint of the robot.
  /// • [6] J7 Seventh joint of the robot, if willbe used.
  SensitivityAxis    : ARRAY[0..6] OF REAL;
  /// Relates to "ThresholdMode" Manual. Defines the threshold of the torque for each robot axis. If the threshold is exceeded, the RA stops.
  /// Index:
  /// • [0] J1 First joint of the robot.
  /// • [1] J2 Second joint of the robot.
  /// • [2] J3 Third joint of the robot.
  /// • [3] J4 Forth joint of the robot.
  /// • [4] J5 Fifth joint of the robot.
  /// • [5] J6 Six joint of the robot.
  /// • [6] J7 Seventh joint of the robot, if will be used
  LimitAxis          : ARRAY[0..6] OF REAL;
  /// Relates to "LimitAxis". Defines the unit of the threshold.
  /// • [0]: Percentage (%) (default) O
  /// • [1]: Newton meter (Nm). O
  /// • [2] Milliampere (mA).
  UnitLimitAxis      : USINT;
  /// Defines the target sequence in which the command will be executed
  SequenceFlag       : SequenceFlag;
END_STRUCT
END_TYPE

{attribute 'pack_mode' := '1'} 
// ------------------------------------------------------------------------- 
//  SRCI Robot Library                                                
// ------------------------------------------------------------------------- 
//                                                                           
//  Object:      CollisionDetectionRecvData                                       
//  Author:      Thorsten Brach                                                
//  Date:        2024-06-22
//
//  Description:                                              
//   
//                                                                           
//  Copyright: 
//    (C) 2024 Thorsten Brach. All rights reserved                                                                                                                                            
//             Licensed under the MIT License.
//                                                                           
//  Disclaimer:                                                                           
//    This project is provided without any guarantee and can be used for   
//    private and commercial purposes. Any use is at the user’s 
//    own risk and responsibility.
//
// -------------------------------------------------------------------------
TYPE CollisionDetectionRecvData EXTENDS RspHeader :
STRUCT
END_STRUCT
END_TYPE

{attribute 'pack_mode' := '1'}
// ------------------------------------------------------------------------- 
//  SRCI Robot Library                                                
// ------------------------------------------------------------------------- 
//                                                                           
//  Object:      CollisionDetectionSendData                                       
//  Author:      Thorsten Brach                                                
//  Date:        2024-06-22
//
//  Description:                                              
//   
//                                                                           
//  Copyright: 
//    (C) 2024 Thorsten Brach. All rights reserved                                                                                                                                            
//             Licensed under the MIT License.
//                                                                           
//  Disclaimer:                                                                           
//    This project is provided without any guarantee and can be used for   
//    private and commercial purposes. Any use is at the user’s 
//    own risk and responsibility.
//
// -------------------------------------------------------------------------
TYPE CollisionDetectionSendData EXTENDS CmdHeader: 
STRUCT
  /// Set TRUE to activate and FALSE to deactivate "CollisionDetection".
  /// Default: TRUE
  ActivateMonitoring : BOOL;
  /// Relates to "LimitAxis". Defines the unit of the threshold.
  /// • [0]: Percentage (%) (default) O
  /// • [1]: Newton meter (Nm). O
  /// • [2] Milliampere (mA).
  UnitLimitAxis      : USINT;
  /// Defines the type of threshold setting (at least one option must be supported)
  ThresholdMode      : ThresholdMode;
  ///  Defines the robot behavior after detecting the collision (at least one option must be supported):
  ReactionMode       : CollisionReactionMode;
  /// Defines the level of sensitivity of all axes.
  /// • 0..99: Sensitivity lower than robot vendor default. 
  ///          At minimum value "0" there is no sensitivity. The lower the value, the lower the sensitivity at the collision detection.
  /// • 100 (default): The value is aligned with the robot vendor-specific default value.
  /// • 101..200: Sensitivity higher than robot vendor default. At maximum value "200" highest possible sensitivity at the collision detection.
  Sensitivity        : INT;
  /// Defines the level of sensitivity of the respective axis.
  /// Values:
  /// • 0..99: Sensitivity lower than robot vendor default. At minimum value "0" there is no sensitivity and collision detection for the respective axis. 
  ///          The lower the value, the lower the sensitivity at the collision detection.
  /// • 100 (default): The value is aligned with the robot vendor-specific default value.
  /// • 101..200: Sensitivity higher than robot vendor default. At maximum value "200" highest possible sensitivity at the collision detection.
  /// Index:
  /// • [0]: J1 First joint of the robot.
  /// • [1]: J2 Second joint of the robot.
  /// • [2] J3 Third joint of the robot.
  /// • [3] J4 Forth joint of the robot.
  /// • [4] J5 Fifth joint of the robot.
  /// • [5] J6 Six joint of the robot.
  /// • [6] J7 Seventh joint of the robot, if willbe used.
  SensitivityAxis    : ARRAY[0..6] OF INT;

  /// Relates to "ThresholdMode" Manual. Defines the threshold of the torque for each robot axis. If the threshold is exceeded, the RA stops.
  /// Index:
  /// • [0] J1 First joint of the robot.
  /// • [1] J2 Second joint of the robot.
  /// • [2] J3 Third joint of the robot.
  /// • [3] J4 Forth joint of the robot.
  /// • [4] J5 Fifth joint of the robot.
  /// • [5] J6 Six joint of the robot.
  /// • [6] J7 Seventh joint of the robot, if will be used
  LimitAxis          : ARRAY[0..6] OF REAL;
END_STRUCT
END_TYPE

{attribute 'pack_mode' := '1'} 
// ------------------------------------------------------------------------- 
//  SRCI Robot Library                                                
// ------------------------------------------------------------------------- 
//                                                                           
//  Object:      ExchangeConfigurationOutCmd                                       
//  Author:      Thorsten Brach                                                
//  Date:        2024-06-22
//
//  Description:                                              
//   
//                                                                           
//  Copyright: 
//    (C) 2024 Thorsten Brach. All rights reserved                                                                                                                                            
//             Licensed under the MIT License.
//                                                                           
//  Disclaimer:                                                                           
//    This project is provided without any guarantee and can be used for   
//    private and commercial purposes. Any use is at the user’s 
//    own risk and responsibility.
//
// -------------------------------------------------------------------------
TYPE ExchangeConfigurationOutCmd :
STRUCT
  /// Returns a metric of how many CMDs it can receive and manage at the same time
  LengthACR                 : UINT;
  /// Highest index of available tools on the RC.
  HighestToolIndex          : USINT;
  /// Highest index of available frames on the RC.
  HighestFrameIndex         : USINT;
  /// Highest index of available loads on the RC.
  HighestLoadIndex          : USINT;
  /// Highest index of available work areas on the RC.
  HighestWorkAreaIndex      : USINT;
  /// Datas which are synchronized
  DataInSync                : DataInSync;
  /// Index of tool changed on RC
  ChangeIndexTool           : USINT;
  /// Index of frame changed on RC
  ChangeIndexFrame          : USINT;
  /// Index of load changed on RC
  ChangeIndexLoad           : USINT;
  ///Index of work area changed on RC
  ChangeIndexWorkArea       : USINT;
  /// Working hours of an RA connected to the RC
  RAWorkingHours            : UDINT;
  /// Signals that a brake test is required in the defined monitoring time (see chapter 6.5.27)
  BrakeTestRequired         : BOOL;
  /// StepMode is active and set to ExactStop (see chapter 6.1.3)
  StepModeExactStopActive   : BOOL;
  /// StepMode is active and set to Blending (see chapter 6.1.3)
  StepModeBlendingActive    : BOOL;
  /// PathAccuracyMode is active (see chapter 6.5.22)
  PathAccuracyMode          : BOOL;
  /// AvoidSingularity is active (see chapter 6.5.23)
  AvoidSingularity          : BOOL;
  /// CollisionDetection is active (see chapter 6.5.35)
  CollisionDetectionEnabled : BOOL;
  /// Cyclic dynamics status bit Accelerating is supported by RC (see chapter 5.5.3.2)
  AcceleratingSupported     : BOOL;
  /// Cyclic dynamics status bit Decelerating is supported by RC (see chapter 5.5.3.2)
  DecceleratingSupported    : BOOL;
  /// Cyclic dynamics status bit ConstantVelocity is supported by RC (see chapter 5.5.3.2)
  ConstantVelocitySupported : BOOL;
  /// Total system hours of an RA connected to the RC. Must not be modifiable by the user.
  /// •  0: Invalid
  /// • >1: Total system hours
  RCWorkingHours            : UDINT;
END_STRUCT
END_TYPE

{attribute 'pack_mode' := '1'} 
// ------------------------------------------------------------------------- 
//  SRCI Robot Library                                                
// ------------------------------------------------------------------------- 
//                                                                           
//  Object:      ExchangeConfigurationParCmd                                       
//  Author:      Thorsten Brach                                                
//  Date:        2024-06-22
//
//  Description:                                              
//   
//                                                                           
//  Copyright: 
//    (C) 2024 Thorsten Brach. All rights reserved                                                                                                                                            
//             Licensed under the MIT License.
//                                                                           
//  Disclaimer:                                                                           
//    This project is provided without any guarantee and can be used for   
//    private and commercial purposes. Any use is at the user’s 
//    own risk and responsibility.
//
// -------------------------------------------------------------------------
TYPE ExchangeConfigurationParCmd :
STRUCT
  /// Defines up to which level of severity messages will be logged in the RC's server log
  LogLevel                   : LogLevel;
  /// Defines blending behavior for single move commands. One of the optional modes must be supported.
  ///  • 0 (default): Move to end position
  ///       Robot moves exactly the target position independently of the selected "BlendingMode"
  ///  • 1: Wait at blending parameter 
  ///       Robot stops its movement when the specified blending parameter is reached
  WaitAtBlendingZone         : BOOL;
  /// Allow a sequence switch from primary to secondary while a subprogram called via CallSubprogram (6.5.18) in the sequence is in progress
  AllowSecSeqWhileSubprogram : BOOL;
  /// Allows blending when CallSubprogram is called in sequence and removed afterwards. For more information see chapter 6.5.21.
  /// • 0 (default): Dynamic blending is prevented
  /// • 1: Dynamic blending is allowed
  AllowDynamicBlending       : BOOL;
  /// Defines waiting time of RC between receiving a first move command when motion queue is empty and starting the first movement. See also chapter 5.6.8.
  DelayTime                  : UINT;
  /// Define number of points required to calculate the blending. See also chapter 5.6.8.
  WaitForNrOfCmd             : UINT;
  /// Maximum allowed time between incrementation of LifeSign before communication error.
  /// • <10 ms: Invalid
  /// • 50 ms: default
  /// See also chapter 5.6.6.2.
  LifeSignTimeOut            : UINT;
  /// Defines a delay time between detecting an inconsistency of configuration data between server and client and executing the defined SyncReaction. 
  /// Always positive. Default: 0 ms
  SyncDelay                  : UINT;
  /// Specifies system reaction in case inconsistency of synchronization data is detected according to Table 6-81. For more information refer to chapter 5.6.7.2
  SyncReaction               : SyncReaction;
  /// Datas which are synchronized
  DataInSync                 : DataInSync;
  /// Enable datas to synchronize
  DataEnableSync             : DataEnableSync;
END_STRUCT
END_TYPE

{attribute 'pack_mode' := '1'} 
// ------------------------------------------------------------------------- 
//  SRCI Robot Library                                                
// ------------------------------------------------------------------------- 
//                                                                           
//  Object:      ExchangeConfigurationRecvData                                       
//  Author:      Thorsten Brach                                                
//  Date:        2024-06-22
//
//  Description:                                              
//   
//                                                                           
//  Copyright: 
//    (C) 2024 Thorsten Brach. All rights reserved                                                                                                                                            
//             Licensed under the MIT License.
//                                                                           
//  Disclaimer:                                                                           
//    This project is provided without any guarantee and can be used for   
//    private and commercial purposes. Any use is at the user’s 
//    own risk and responsibility.
//
// -------------------------------------------------------------------------
TYPE ExchangeConfigurationRecvData EXTENDS RspHeader :
STRUCT
  /// TRUE when function is exchanging data
  Enabled                   : BOOL;
  /// Reserve 
  Reserve1                  : BYTE;
   /// Returns a metric of how many CMDs it can receive and manage at the same time
  LengthACR                 : UINT;
  /// Highest index of available tools on the RC.
  HighestToolIndex          : USINT;
  /// Highest index of available frames on the RC.
  HighestFrameIndex         : USINT;
  /// Highest index of available loads on the RC.
  HighestLoadIndex          : USINT;
  /// Highest index of available work areas on the RC.
  HighestWorkAreaIndex      : USINT; 
  /// Datas which are synchronized
  DataInSync                : DataInSync;
  /// Reserve 
  Reserve2                  : BYTE;
  /// Index of tool changed on RC
  ChangeIndexTool           : USINT;
  /// Index of frame changed on RC
  ChangeIndexFrame          : USINT;
  /// Index of load changed on RC
  ChangeIndexLoad           : USINT;
  ///Index of work area changed on RC
  ChangeIndexWorkArea       : USINT;
  /// Working hours of an RA connected to the RC
  RAWorkingHours            : UDINT;
  /// Status byte
  StatusByte                : BYTE;
  /// Cyclic dynamics status bit ConstantVelocity is supported by RC (see chapter 5.5.3.2)
  ConstantVelocitySupported : BOOL;
  /// Total system hours of an RA connected to the RC. Must not be modifiable by the user.
  /// •  0: Invalid
  /// • >1: Total system hours
  RCWorkingHours            : UDINT;
END_STRUCT
END_TYPE

{attribute 'pack_mode' := '1'}
// ------------------------------------------------------------------------- 
//  SRCI Robot Library                                                
// ------------------------------------------------------------------------- 
//                                                                           
//  Object:      ExchangeConfigurationSendData                                       
//  Author:      Thorsten Brach                                                
//  Date:        2024-06-22
//
//  Description:                                              
//   
//                                                                           
//  Copyright: 
//    (C) 2024 Thorsten Brach. All rights reserved                                                                                                                                            
//             Licensed under the MIT License.
//                                                                           
//  Disclaimer:                                                                           
//    This project is provided without any guarantee and can be used for   
//    private and commercial purposes. Any use is at the user’s 
//    own risk and responsibility.
//
// -------------------------------------------------------------------------
TYPE ExchangeConfigurationSendData EXTENDS CmdHeader: 
STRUCT
  /// Defines up to which level of severity messages will be logged in the RC's server log
  LogLevel                   : LogLevel;
  /// Miscellaneous control bits 
  CtrlByte                   : BYTE;
  /// Defines waiting time of RC between receiving a first move command when motion queue is empty and starting the first movement. See also chapter 5.6.8.
  DelayTime                  : UINT;
  /// Define number of points required to calculate the blending. See also chapter 5.6.8.
  WaitForNrOfCmd             : UINT;
  /// Maximum allowed time between incrementation of LifeSign before communication error.
  /// • <10 ms: Invalid
  /// • 50 ms: default
  /// See also chapter 5.6.6.2.
  LifeSignTimeOut            : UINT;
  /// Defines a delay time between detecting an inconsistency of configuration data between server and client and executing the defined SyncReaction. 
  /// Always positive. Default: 0 ms
  SyncDelay                  : UINT;
  /// Specifies system reaction in case inconsistency of synchronization data is detected according to Table 6-81. For more information refer to chapter 5.6.7.2
  SyncReaction               : SyncReaction;
  /// Reserve
  Reserve1                    : BYTE; // bth3ho fanuc
  /// Datas which are synchronized
  DataInSync                 : DataInSync;
  /// Reserve
  Reserve2                   : BYTE;
  /// Enable datas to synchronize
  DataEnableSync             : DataEnableSync;  
  /// Reserve
  Reserve3                   : BYTE;
END_STRUCT
END_TYPE

{attribute 'pack_mode' := '1'} 
// ------------------------------------------------------------------------- 
//  SRCI Robot Library                                                
// ------------------------------------------------------------------------- 
//                                                                           
//  Object:      FreeDriveOutCmd                                       
//  Author:      Thorsten Brach                                                
//  Date:        2024-06-22
//
//  Description:                                              
//   
//                                                                           
//  Copyright: 
//    (C) 2024 Thorsten Brach. All rights reserved                                                                                                                                            
//             Licensed under the MIT License.
//                                                                           
//  Disclaimer:                                                                           
//    This project is provided without any guarantee and can be used for   
//    private and commercial purposes. Any use is at the user’s 
//    own risk and responsibility.
//
// -------------------------------------------------------------------------
TYPE FreeDriveOutCmd :
STRUCT
  /// TRUE while "FreeDrive" is active.
  Enabled : BOOL;
END_STRUCT
END_TYPE

